// TIA Portal V19 export
DATA_BLOCK "ControlNodes"   // DB76
// stored: Access Published, MemoryReserve 100, Namespace Unit3.EM1
   VAR
      em { ExternalWritable := 'False'} : "LAF_typeEmControlNode";
      jobs { ExternalWritable := 'False'} : "LAF_typeJobs";
      sequence { ExternalWritable := 'False'} : "LAF_typeSequence";
      cm1SignalTm { S7_SetPoint := 'True'} : "EXCHANGETRAY_typeNgConveyorIoSignalControlNode";
      cm2AxisControl : "LBC_typeAxisSimpleControlNode_1";
      cm3NgStrapPositionDetection : "LEXCHANGETRAY_typeNgStrapControlNode";
      cm4FrButton { S7_SetPoint := 'True'} : "EXCHANGETRAY_typeFrButtonControlNode";
      jobConditions : "Unit3.EM1.ZSL_typeJobConditionsControlNode";
   END_VAR
BEGIN
   em.status.enabled := true;
END_DATA_BLOCK
